{attribute 'qualified_only'}
{attribute 'strict'}
TYPE eOverallResult : 
(
    NoAction := 0,
    InProgress := 10,
    Passed := 20,
    Failed := 30
);
END_TYPE

(* stored: Version 1.1.0.1, ProductVersion 3.1.4024.9
   DUT eOverallResult: Id {01216d0c-dd53-0320-2aac-4d70b3767dc4} *)
